// Mitsubishi GX Works2 project: plcbitword   PLC: Q03UDV

PROGRAM MAIN
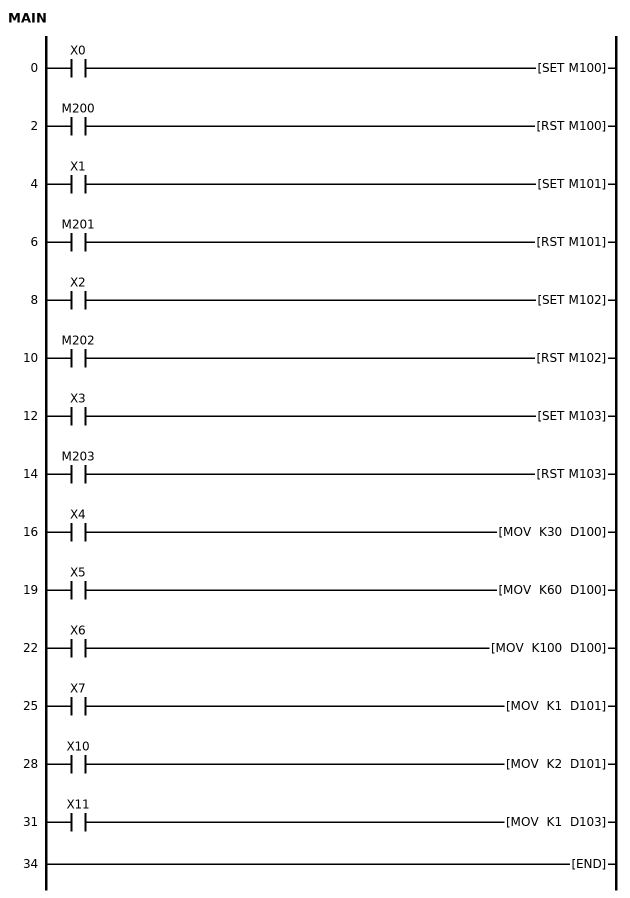
0     LD      X0
      SET     M100
2     LD      M200
      RST     M100
4     LD      X1
      SET     M101
6     LD      M201
      RST     M101
8     LD      X2
      SET     M102
10    LD      M202
      RST     M102
12    LD      X3
      SET     M103
14    LD      M203
      RST     M103
16    LD      X4
      MOV     K30 D100
19    LD      X5
      MOV     K60 D100
22    LD      X6
      MOV     K100 D100
25    LD      X7
      MOV     K1 D101
28    LD      X10
      MOV     K2 D101
31    LD      X11
      MOV     K1 D103
34    END
END_PROGRAM
